FUNCTION_BLOCK FB_Module_CoilPusher IMPLEMENTS I_Module
VAR_INPUT
	bEnable		: BOOL;
END_VAR
VAR_OUTPUT
END_VAR
VAR
	Components	: ARRAY [0..1] OF I_Component;
	
	fbServo		: FB_Component_ServoMotor;
	fbSensor	: FB_Component_InductiveSensor;
	
	idx			: INT;
END_VAR

IF bEnable THEN
	fbServo(
		bEnable 			:= TRUE, 
		bHomingSensor 		:= GVL.bCoilTranslate, 
		bHomingSpeed 		:= 0, 
		uMaxRPM 			:= 3000,
		bSetCounterDone		:= GVL.bSetCounterDoneServo1,
		rGearRatio			:= 1,
		dCountServo			:= GVL.dCountServo1,
		bSetCounter			:= GVL.dSetCounterServo1,
		dSetCounterValue	:= GVL.dSetCounterValueServo1,
		bEnableDrive 		:= GVL.b603Enable, 
		uAnalogOut 			:= GVL.aOutServo1);
	
	fbSensor(
		bRawSignal			:= GVL.bCoilTranslate,
		tDebounce			:= T#5MS,
		tTimeout			:= T#5MS,
		sName				:= 'translate coil sens',
		bEnable				:= TRUE);
	
	Components[0]	:= fbServo;
	Components[1]	:= fbSensor;
	
	FOR idx := 0 TO 1 DO
    	Components[idx].M_Start();
	END_FOR;
END_IF

METHOD M_Extend : BOOL
VAR_INPUT
	uPos	: INT;
END_VAR
IF bEnable THEN
	M_Extend := fbServo.M_Goto(30000, 2, 500);
END_IF
END_METHOD

{warning 'add method implementation '}
METHOD M_Halt : BOOL
END_METHOD

METHOD M_Home : BOOL
VAR_INPUT
END_VAR
IF bEnable THEN
	IF fbSensor.bSensorActive THEN
		fbServo.M_SetSpeed(0);
		fbServo.M_DisableDrive();
		IF fbServo.M_SetCounter(0) THEN
			M_Home := TRUE;
		END_IF
	ELSE
		fbServo.M_EnableDrive();
		fbServo.M_SetSpeed(-2);
	END_IF
END_IF
END_METHOD

{warning 'add method implementation '}
METHOD M_Start : BOOL
END_METHOD

{warning 'add method implementation '}
METHOD M_Stop : BOOL
END_METHOD

END_FUNCTION_BLOCK

(* stored: Version 1.1.0.1, ProductVersion 3.1.4024.15
   POU FB_Module_CoilPusher: Id {8e8d1dee-ebd9-4fec-b79d-3fb510dceae4}, SpecialFunc None
   Method M_Extend: Id {2b1df13a-2b1d-4b0a-acb6-5cb20add145c}
   Method M_Halt: Id {58ed4357-7aac-4b0b-a942-3662baab7bcf}
   Method M_Home: Id {2547e027-85d7-4928-ad7f-ba321c02857c}
   Method M_Start: Id {5de6f7fa-b867-4cfe-b380-2067954c8bd8}
   Method M_Stop: Id {33e9907a-70e6-4926-9b25-8911ec5525b0} *)
